{attribute 'Tc2GvlVarNames'}
VAR_GLOBAL CONSTANT
END_VAR

(* stored: Version 1.1.0.1, ProductVersion 3.1.4022.7
   GVL Constants: Id {127c0793-6509-4d62-a07d-391d2fb3f0a9} *)
